// TIA Portal V19 export
VAR_GLOBAL   // PLC tag table "KP8Tags"
   Toggle_Switch2 AT %M50.0 : Bool;   // KP8 bit that is toggled each time is pressed
   HMI_KP8_JogFwd AT %M50.1 : Bool;
   HMI_KP8_Stop AT %M50.2 : Bool;
   Toggle_Switch1 AT %M50.4 : Bool;   // KP8 bit that is toggled each time is pressed
   HMI_KP8_JogRev AT %M50.5 : Bool;
   HMI_KP8_Start AT %M50.6 : Bool;
   Toggle_Enable_Disable AT %M50.7 : Bool;   // KP8 bit that is toggled each time is pressed
   HMI_KP8_Red AT %MB70 : Byte;
   HMI_KP8_Green AT %MB71 : Byte;
   HMI_KP8_Blue AT %MB72 : Byte;
   HMI_KP8_Enable_Disable AT %M73.0 : Bool;
   HMI_KP8_Reset AT %M73.1 : Bool;
   HMI_KP8_Switch1 AT %M73.2 : Bool;
   HMI_KP8_Switch2 AT %M73.3 : Bool;
   OS8 AT %M74.0 : Bool;
   OS9 AT %M74.1 : Bool;
   OS10 AT %M74.2 : Bool;
END_VAR
